INTERFACE I_PrintGlobal

PROPERTY iHardwarePool : I_HardwarePool
GET
END_GET
END_PROPERTY

PROPERTY iMasterPrintPosition : I_PrintPosition
GET
END_GET
END_PROPERTY

(*
  Register for PU StatusClient
*)
METHOD registerPuStatusClient : BOOL
VAR_INPUT
  sClient       : I_PrintStatusClient;
END_VAR
END_METHOD

METHOD registerPuSubystem : BOOL
VAR_INPUT
  iSubSys      : I_PrintSubsystem;
END_VAR
END_METHOD

END_INTERFACE

(* stored: Version 1.1.0.1, ProductVersion 3.1.4024.11
   Itf I_PrintGlobal: Id {21c90071-c4b1-47be-a0ad-3c64a278d0e6}
   Property iHardwarePool: Id {b6d2dee3-9f7c-4dc8-a78b-294dfdcc87ad}
   Get Get: Id {37d2349b-3cf6-4a81-9de1-4be811653e6e}
   Property iMasterPrintPosition: Id {ebb31c12-29b2-4913-828d-32887cc26ddb}
   Get Get: Id {cfa54b9f-29fd-4e1d-a222-ac56e5623fab}
   Method registerPuStatusClient: Id {c83083f8-aed4-490c-ab6f-30bf48136e4a}
   Method registerPuSubystem: Id {bc9e8bd5-c97d-4bef-a418-ad671ac1dd5b} *)
